(* Logix 5000 project; controller PLC_FANUC vendor 1 type 14 code 226 rev 35.11; software revision 35.00 *)

TASK MainTask (continuous, watchdog 500 ms) : MainProgram
TASK SafetyTask (periodic, rate 20 ms, priority 10, watchdog 20 ms, safety) : SafetyProgram

MODULES
   Local : vendor 1 type 14 code 226 (5069 0, rev 35.11)
      Robot : ETHERNET-MODULE (Ethernet 10.32.81.61, rev 1.1, Output RPI 30 ms)
           Robot:I.Data[1].4   // CMD Enabled
           Robot:I.Data[1].5   // System Ready
           Robot:I.Data[1].6   // Program Running
           Robot:I.Data[1].7   // Program Paused
           Robot:I.Data[1].8   // Motion Held
           Robot:I.Data[1].9   // Fault
           Robot:I.Data[1].10   // At Perch
           Robot:I.Data[1].11   // TP Enabled
           Robot:O.Data[1].4   // IMSTP
           Robot:O.Data[1].5   // Hold
           Robot:O.Data[1].6   // SFSPD
           Robot:O.Data[1].7   // Cycle Stop
           Robot:O.Data[1].8   // Fault Reset
           Robot:O.Data[1].9   // Start
           Robot:O.Data[1].10   // Home
           Robot:O.Data[1].11   // Enabled
           Robot:O.Data[1].12   // DI-101
       : 5069-OB16 (5069 2, rev 1.50, StandardDataDriven RPI 5 ms)
       : 5069-IB16 (5069 1, rev 1.50, StandardDataDriven RPI 5 ms)
           Local:1:I.Pt03.Data   // Light Curtain
END_MODULES

PROGRAM MainProgram   (* main routine MainRoutine *)
VAR
   enable : BOOL;
   fault : BOOL;
   FirstTimer : TIMER := (PRE := 1100);
   safe : BOOL;
   SecondTimer : TIMER := (PRE := 1100);
   start : BOOL;
   StartAir : BOOL;
   StartButton : BOOL;
   StartProgram : BOOL;
   stop : BOOL;
   StopAir : BOOL;
   SwapAir : BOOL;
   WaitTillDone1 : BOOL;
   WaitTillDone2 : BOOL;
END_VAR

ROUTINE MainRoutine   (* ladder *)
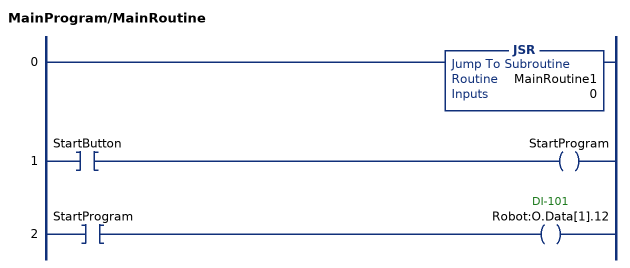
   0: JSR(MainRoutine1,0);
   1: XIC(StartButton)OTE(StartProgram);
   2: XIC(StartProgram)OTE(Robot:O.Data[1].12);
END_ROUTINE

ROUTINE MainRoutine1   (* ladder *)
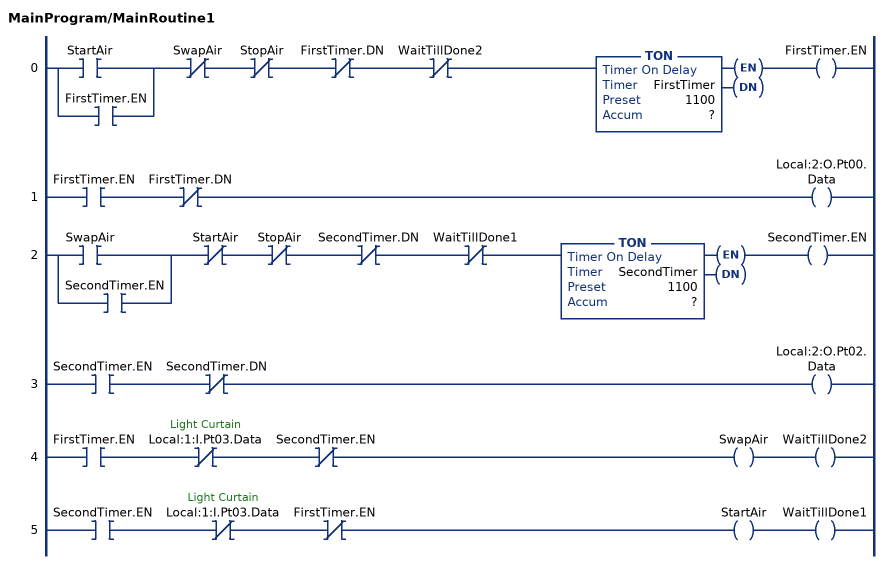
   0: [XIC(StartAir) ,XIC(FirstTimer.EN) ]XIO(SwapAir)XIO(StopAir)XIO(FirstTimer.DN)XIO(WaitTillDone2)TON(FirstTimer,?,?)OTE(FirstTimer.EN);
   1: XIC(FirstTimer.EN)XIO(FirstTimer.DN)OTE(Local:2:O.Pt00.Data);
   2: [XIC(SwapAir) ,XIC(SecondTimer.EN) ]XIO(StartAir)XIO(StopAir)XIO(SecondTimer.DN)XIO(WaitTillDone1)TON(SecondTimer,?,?)OTE(SecondTimer.EN);
   3: XIC(SecondTimer.EN)XIO(SecondTimer.DN)OTE(Local:2:O.Pt02.Data);
   4: XIC(FirstTimer.EN)XIO(Local:1:I.Pt03.Data)XIO(SecondTimer.EN)OTE(SwapAir)OTE(WaitTillDone2);
   5: XIC(SecondTimer.EN)XIO(Local:1:I.Pt03.Data)XIO(FirstTimer.EN)OTE(StartAir)OTE(WaitTillDone1);
END_ROUTINE
END_PROGRAM

PROGRAM SafetyProgram   (* main routine MainRoutine, safety *)

ROUTINE MainRoutine   (* ladder *)
   0 (stored rung type 13): ;
END_ROUTINE
END_PROGRAM
